FUNCTION_BLOCK ABSTRACT TaskBase IMPLEMENTS ITask
VAR
	_busy : BOOL;
	_error : BOOL;
	_done : BOOL;
	State: INT;
END_VAR

METHOD Abort : BOOL
VAR_INPUT
END_VAR
END_METHOD

PROPERTY Busy : BOOL
GET
Busy := _busy;
END_GET
END_PROPERTY

PROPERTY Done : BOOL
GET
Done := _done;
END_GET
END_PROPERTY

PROPERTY Error : BOOL
GET
Error := _error;
END_GET
END_PROPERTY

END_FUNCTION_BLOCK

(* stored: Version 1.1.0.1, ProductVersion 3.1.4024.12
   POU TaskBase: Id {fbf26ffd-7a30-4e38-9264-b2fd1838bbf2}, SpecialFunc None
   Method Abort: Id {6b87c897-5db6-41a6-afc4-56be8a5c8140}
   Property Busy: Id {f43d865a-539d-4bae-9ff8-de21a1fd6356}
   Get Get: Id {0f53bcc7-4c05-4a35-b63a-3d4286c0d863}
   Property Done: Id {b91c8789-596c-4b5e-b921-d7d4df7c5752}
   Get Get: Id {50d6abe5-34d8-47af-944c-254d2cc6a361}
   Property Error: Id {7ac774a4-60d3-43cf-a9cd-482a5232e7e0}
   Get Get: Id {4085b453-daf4-4126-8576-5e320e3e1f25} *)
